// TIA Portal V20 export
TYPE "LKinCtrl_typePnPOrientationFrame"
   STRUCT
      "a" : LReal;   // Orientation A
      "b" : LReal;   // Orientation B
      c : LReal;   // Orientation C
   END_STRUCT;
END_TYPE
